TYPE T_CodeMRP : STRING[8];
END_TYPE

(* stored: Version 1.1.0.1
   DUT T_CodeMRP: Id {5b364791-20ae-41ce-8f0e-822b94ac97e0} *)
